Yaskawa INFORM job: test1TRJ0.JBI

/JOB
//NAME test1TRJ0
//POS
///NPOS 5,0,0,0,0,0
///TOOL 1
///POSTYPE ROBOT
///RECTAN
///RCONF 1,0,0,0,0,0,0,0,0,0,0,0,0,0,0,0,0,0,0,0,0,0,0,0
C00000=0.000,=0.000,=0.000,=1.0000,=0.0,=0.0000
C00001=10.000,=10.000,=10.000,=0.0000,=1.0,=0.0000
C00002=20.000,=20.000,=20.000,=0.0000,=0.0,=1.0000
C00003=30.000,=30.000,=30.000,=1.0000,=0.0,=0.0000
C00004=40.000,=40.000,=40.000,=1.0000,=0.0,=0.0000
//INST
///DATE 2021/02/10 13:51
///COMM
///ATTR SC,RW,RJ
////FRAME USER 2
///GROUP1 RB1
NOP
' first example of file for tool generation
SPEED V=10.2
MOVL C00001
SPEED V=50.0
MOVL C00002
MOVL C00003
TIMER T=10.23
DOUT OG#(12) 1
ARCON
MOVL C00004
ARCOF
MOVL C00005
END
